// SIMATIC S7-200 project (STEP 7-Micro/WIN), CPU 224XP REL 02.01

ORGANIZATION_BLOCK MAIN:OB1
TITLE=PROGRAM COMMENTS
BEGIN
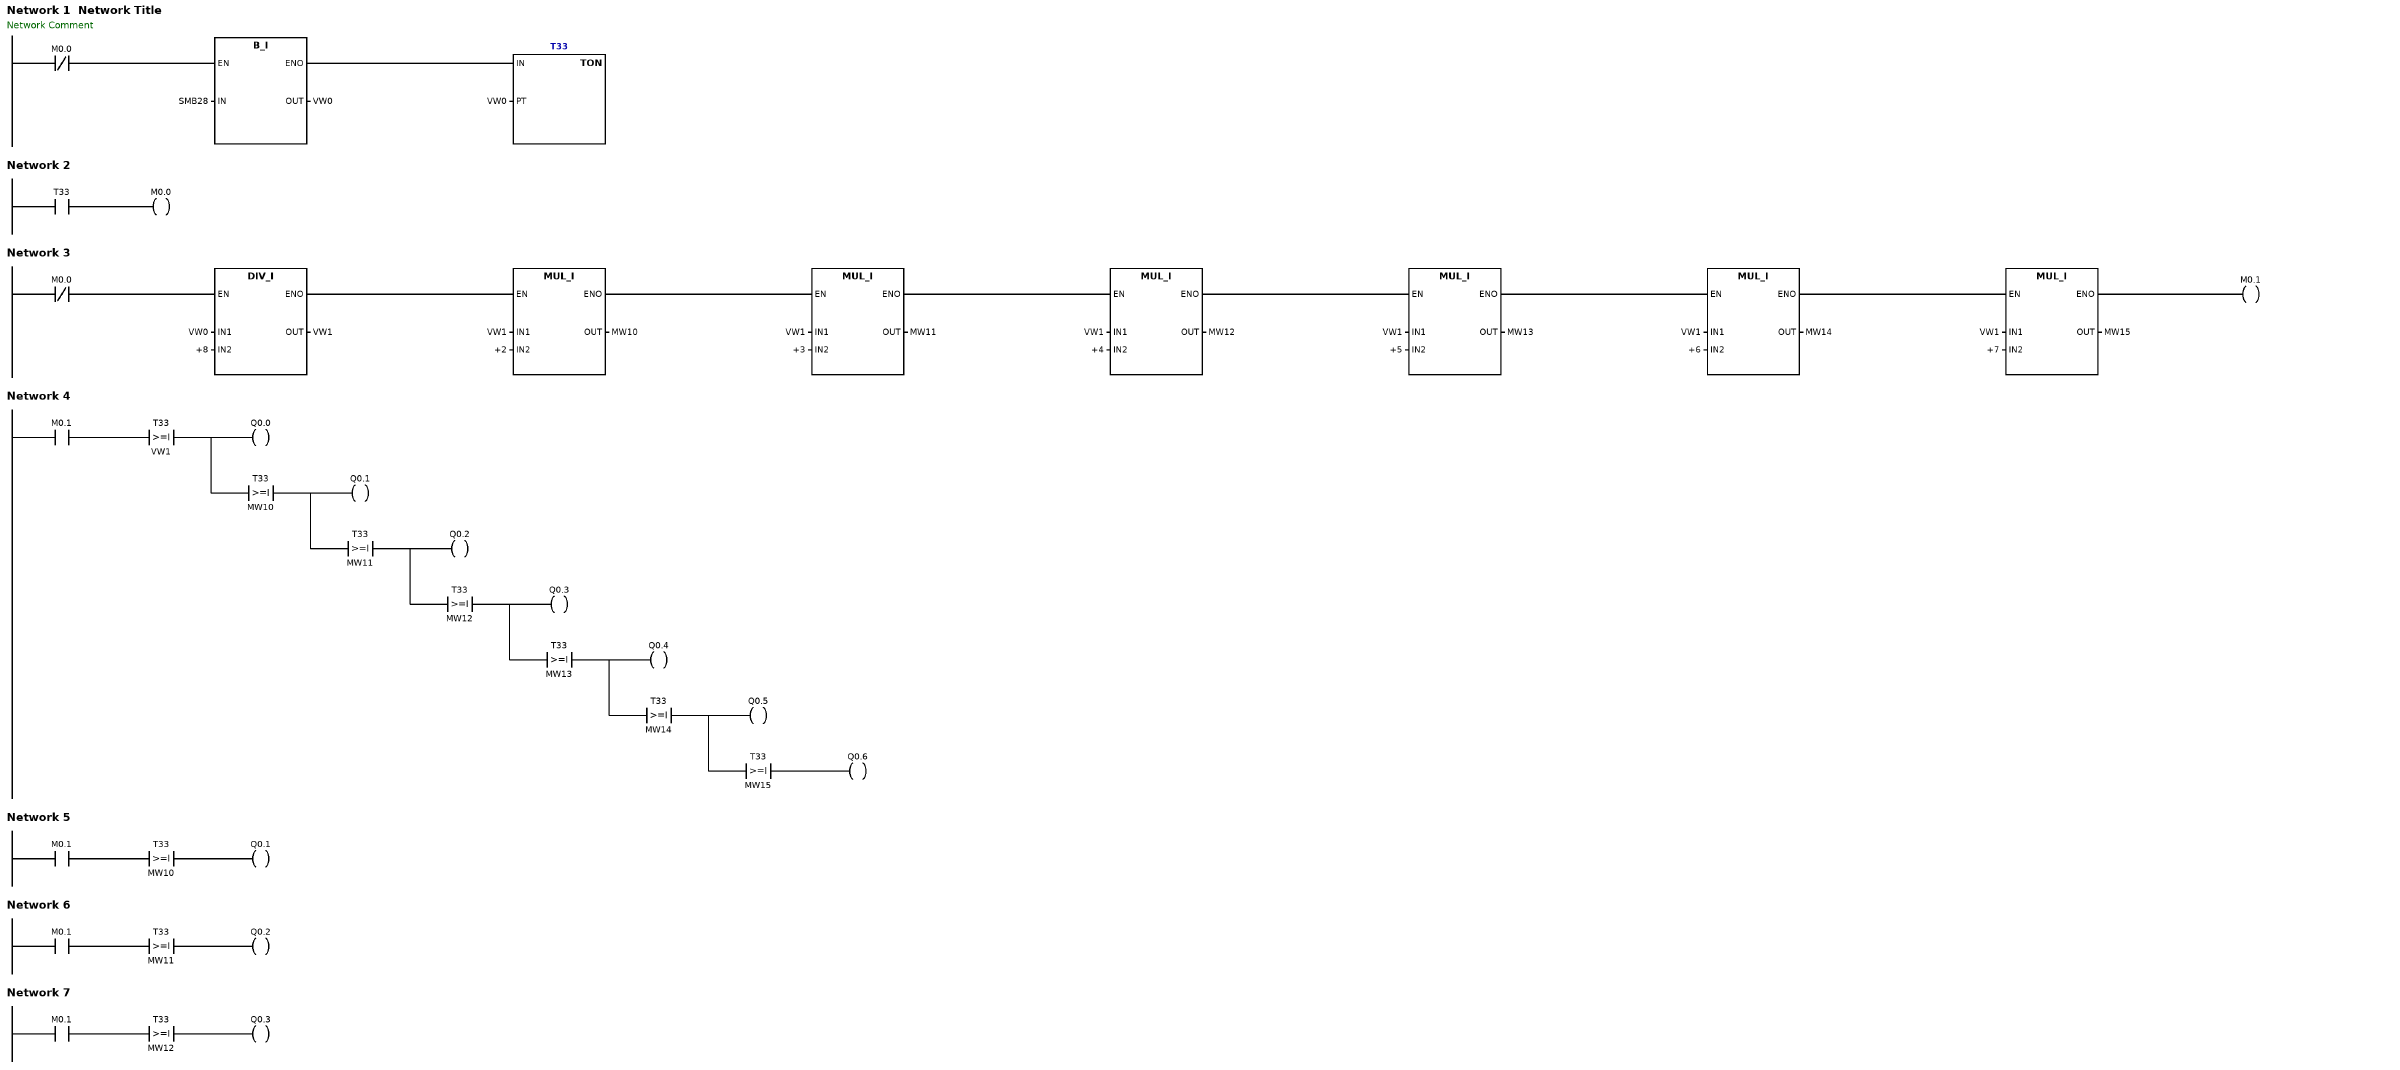
Network 1 // Network Title
// Network Comment
LDN    M0.0
BTI    SMB28, VW0
AENO
TON    T33, VW0
Network 2
LD     T33
=      M0.0
Network 3
LDN    M0.0
MOVW   VW0, VW1
AENO
/I     +8, VW1
AENO
MOVW   VW1, MW10
AENO
*I     +2, MW10
AENO
MOVW   VW1, MW11
AENO
*I     +3, MW11
AENO
MOVW   VW1, MW12
AENO
*I     +4, MW12
AENO
MOVW   VW1, MW13
AENO
*I     +5, MW13
AENO
MOVW   VW1, MW14
AENO
*I     +6, MW14
AENO
MOVW   VW1, MW15
AENO
*I     +7, MW15
AENO
=      M0.1
Network 4
// (network saved uncompiled; LAD cells follow)
// row 0: c0 -| |- M0.1  c1 -|>=I|- T33, VW1 v  c2 -( ) Q0.0
// row 1: c1 ^  c2 -|>=I|- T33, MW10 v  c3 -( ) Q0.1
// row 2: c2 ^  c3 -|>=I|- T33, MW11 v  c4 -( ) Q0.2
// row 3: c3 ^  c4 -|>=I|- T33, MW12 v  c5 -( ) Q0.3
// row 4: c4 ^  c5 -|>=I|- T33, MW13 v  c6 -( ) Q0.4
// row 5: c5 ^  c6 -|>=I|- T33, MW14 v  c7 -( ) Q0.5
// row 6: c6 ^  c7 -|>=I|- T33, MW15  c8 -( ) Q0.6
Network 5
// (network saved uncompiled; LAD cells follow)
// row 0: c0 -| |- M0.1  c1 -|>=I|- T33, MW10  c2 -( ) Q0.1
Network 6
// (network saved uncompiled; LAD cells follow)
// row 0: c0 -| |- M0.1  c1 -|>=I|- T33, MW11  c2 -( ) Q0.2
Network 7
// (network saved uncompiled; LAD cells follow)
// row 0: c0 -| |- M0.1  c1 -|>=I|- T33, MW12  c2 -( ) Q0.3
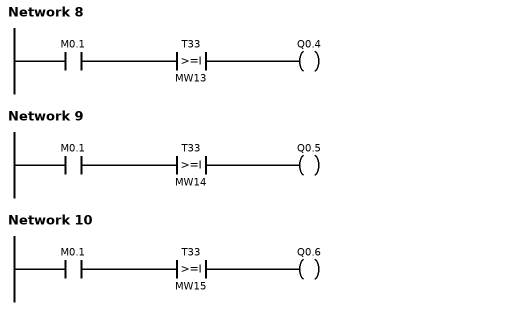
Network 8
// (network saved uncompiled; LAD cells follow)
// row 0: c0 -| |- M0.1  c1 -|>=I|- T33, MW13  c2 -( ) Q0.4
Network 9
// (network saved uncompiled; LAD cells follow)
// row 0: c0 -| |- M0.1  c1 -|>=I|- T33, MW14  c2 -( ) Q0.5
Network 10
// (network saved uncompiled; LAD cells follow)
// row 0: c0 -| |- M0.1  c1 -|>=I|- T33, MW15  c2 -( ) Q0.6
END_ORGANIZATION_BLOCK
